// TIA Portal V17 export
// export: Created 2022-11-28T05:31:03.7953951Z, ExportSetting WithDefaults, DisplayName Totally Integrated Automation Portal, DisplayVersion V17, DisplayName TIA Portal Openness, DisplayVersion V17, DisplayName TIA Portal Version Control Interface, DisplayVersion V17, DisplayName STEP 7 Professional, DisplayVersion V17, DisplayName STEP 7 Safety, DisplayVersion V17, DisplayName WinCC Professional, DisplayVersion V17
FUNCTION_BLOCK "MultiProcessing_FB"   // FB2, LAD
{ S7_Optimized_Access := 'TRUE' }
VERSION : 0.1
// stored: AutoNumber true, IsIECCheckEnabled false, IsRetainMemResEnabled false, MemoryReserve 100, SetENOAutomatically false, UDAEnableTagReadback false
   VAR_INPUT
      Start : Bool;
      Reset : Bool;
      RefSwitchTurnTable_PosVac : Bool;
      RefSwitchTurnTable_PosBelt : Bool;
      RefSwitchTurnTable_PosSaw : Bool;
      RefSwitchVac_PosTurnTable : Bool;
      RefSwitchVac_PosOven : Bool;
      RefSwitchOven_FeederInside : Bool;
      RefSwitchOven_FeederOutside : Bool;
      LightBarrierOven : Bool;
      LightBarrierEndOfConBelt : Bool;
   END_VAR
   VAR_OUTPUT
      M2_ConveyorBeltForward : Bool;
      M3_Saw : Bool;
      M4_OvenFeederRetract : Bool;
      M4_OvenFeederExtend : Bool;
      LightOven : Bool;
      PWM_TurnTable : Int;
      PWM_Vacuum : Int;
      Compressor : Bool := true;
   END_VAR
   VAR_IN_OUT
      M1_TurnTableClockwise : Bool;
      M1_TurnTableCounterclockwise : Bool;
      M5_VacuumTowardsOven : Bool;
      M5_VacuumTowardsTurnTable : Bool;
      ValveVacuum : Bool;
      ValveLowering : Bool;
      ValveOvenDoor : Bool;
      ValveFeeder : Bool;
   END_VAR
   VAR
      FeederLoaded : Bool;
      Step_Oven : Int := 0;
      Step_Vacuum : Int := 0;
      Step_TurnTable : Int := 0;
      OpenOvenDoor0 : Bool;
      OpenOvenDoor1 : Bool;
      OpenOvenDoor2 : Bool;
      CloseOvenDoor : Bool;
      Lower0 : Bool;
      Lower1 : Bool;
      Rise0 : Bool;
      Rise1 : Bool;
      Rise2 : Bool;
      M2_TurnTableClockwise : Bool;
      M3_TurnTableClockwise : Bool;
      ActivateVacuum0 : Bool;
      ActivateVacuum1 : Bool;
      DeactivateVacuum : Bool;
      IEC_Timer_LoweringDown { S7_SetPoint := 'True'} : IEC_TIMER;
      IEC_Timer_VacuumOn { S7_SetPoint := 'True'} : IEC_TIMER;
      IEC_Timer_LoweringUp { S7_SetPoint := 'True'} : IEC_TIMER;
      IEC_Timer_VacuumOff { S7_SetPoint := 'True'} : IEC_TIMER;
      IEC_Timer_OvenClose { S7_SetPoint := 'True'} : IEC_TIMER;
      IEC_Timer_OvenLight { S7_SetPoint := 'True'} : IEC_TIMER;
      IEC_Timer_OvenOpen { S7_SetPoint := 'True'} : IEC_TIMER;
      IEC_Timer_Saw { S7_SetPoint := 'True'} : IEC_TIMER;
      IEC_Timer_Onloading { S7_SetPoint := 'True'} : TON_TIME;
      IEC_Timer_Offloading { S7_SetPoint := 'True'} : TON_TIME;
      IEC_Timer_LoweringDownOnOven { S7_SetPoint := 'True'} : TON_TIME;
      IEC_Timer_LoweringUpOffOven { S7_SetPoint := 'True'} : TON_TIME;
      IEC_Timer_OvenReset { S7_SetPoint := 'True'} : TON_TIME;
      IEC_Timer_TurnTablePush { S7_SetPoint := 'True'} : TON_TIME;
      IEC_Timer_DeactivateConveyorBelt { S7_SetPoint := 'True'} : TOF_TIME;
      IEC_Timer_0_Instance { S7_SetPoint := 'True'} : TOF_TIME;
   END_VAR
   VAR_TEMP   // added for the SCL form of the ladder/FBD networks
      _w1 : Bool;
   END_VAR
BEGIN

REGION Network 1: Start/Stop
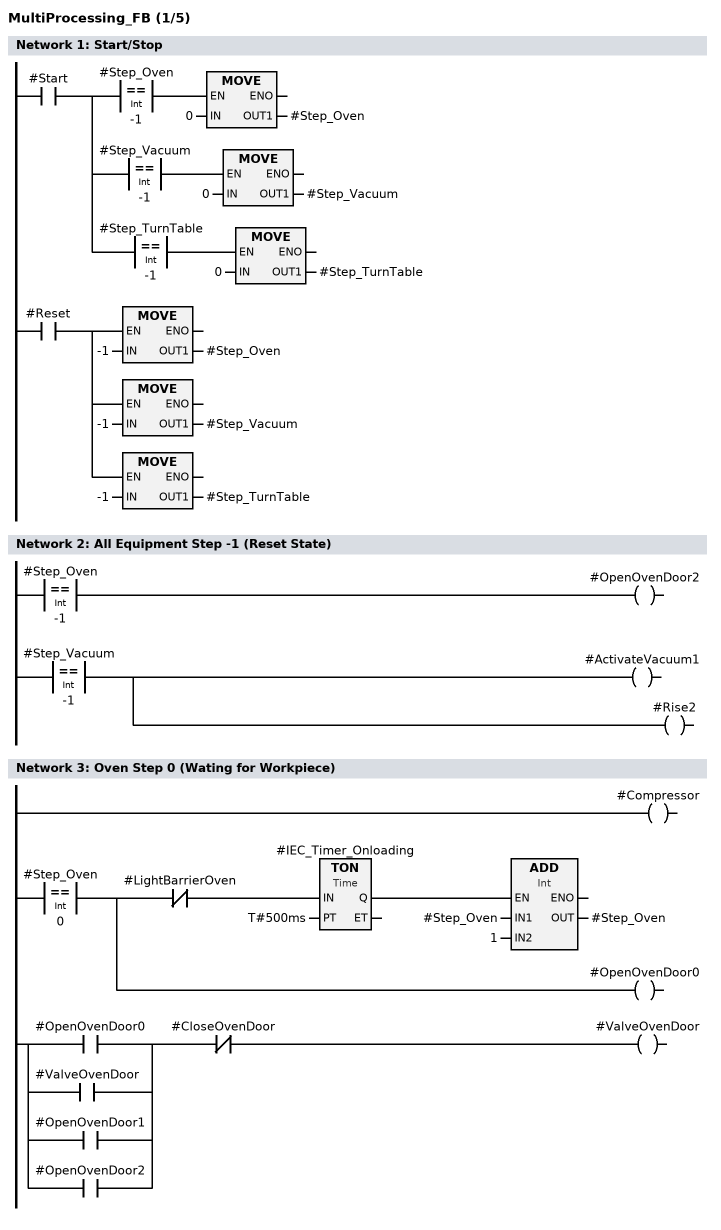
   RUNG wire#powerrail
      Contact( #Start )
      wire#w1
      { S7_Templates := "SrcType := Int" } EQ_Contact(in1 := #Step_Oven, in2 := -1)
      Move(in := 0, out1 => #Step_Oven)
   END_RUNG
   RUNG wire#w1
      { S7_Templates := "SrcType := Int" } EQ_Contact(in1 := #Step_Vacuum, in2 := -1)
      Move(in := 0, out1 => #Step_Vacuum)
   END_RUNG
   RUNG wire#w1
      { S7_Templates := "SrcType := Int" } EQ_Contact(in1 := #Step_TurnTable, in2 := -1)
      Move(in := 0, out1 => #Step_TurnTable)
   END_RUNG
   RUNG wire#powerrail
      Contact( #Reset )
      wire#w2
      Move(in := -1, out1 => #Step_Oven)
   END_RUNG
   RUNG wire#w2
      Move(in := -1, out1 => #Step_Vacuum)
   END_RUNG
   RUNG wire#w2
      Move(in := -1, out1 => #Step_TurnTable)
   END_RUNG
   // the same network as SCL:
   IF #Start AND (#Step_Oven = (-1)) THEN #Step_Oven := 0; END_IF;
   IF #Start AND (#Step_Vacuum = (-1)) THEN #Step_Vacuum := 0; END_IF;
   IF #Start AND (#Step_TurnTable = (-1)) THEN #Step_TurnTable := 0; END_IF;
   IF #Reset THEN
       #Step_Oven := -1;
       #Step_Vacuum := -1;
       #Step_TurnTable := -1;
   END_IF;
END_REGION

REGION Network 2: All Equipment Step -1 (Reset State)
   RUNG wire#powerrail
      { S7_Templates := "SrcType := Int" } EQ_Contact(in1 := #Step_Oven, in2 := -1)
      Coil( #OpenOvenDoor2 )
   END_RUNG
   RUNG wire#powerrail
      { S7_Templates := "SrcType := Int" } EQ_Contact(in1 := #Step_Vacuum, in2 := -1)
      wire#w1
      Coil( #ActivateVacuum1 )
   END_RUNG
   RUNG wire#w1
      Coil( #Rise2 )
   END_RUNG
   // the same network as SCL:
   #OpenOvenDoor2 := #Step_Oven = (-1);
   #ActivateVacuum1 := #Step_Vacuum = (-1);
   #Rise2 := #ActivateVacuum1;
END_REGION

REGION Network 3: Oven Step 0 (Wating for Workpiece)
   RUNG wire#powerrail
      Coil( #Compressor )
   END_RUNG
   RUNG wire#powerrail
      { S7_Templates := "SrcType := Int" } EQ_Contact(in1 := #Step_Oven, in2 := 0)
      wire#w1
      I_Contact( #LightBarrierOven )
      { S7_Templates := "time_type := Time" } #IEC_Timer_Onloading.TON(pt := T#500ms, et =>)
      { S7_Templates := "SrcType := Int" } Add(in1 := #Step_Oven, in2 := 1, out => #Step_Oven)
   END_RUNG
   RUNG wire#w1
      Coil( #OpenOvenDoor0 )
   END_RUNG
   RUNG wire#powerrail
      Contact( #OpenOvenDoor0 )
      wire#w2
      I_Contact( #CloseOvenDoor )
      Coil( #ValveOvenDoor )
   END_RUNG
   RUNG wire#powerrail
      Contact( #ValveOvenDoor )
   END_RUNG wire#w2
   RUNG wire#powerrail
      Contact( #OpenOvenDoor1 )
   END_RUNG wire#w2
   RUNG wire#powerrail
      Contact( #OpenOvenDoor2 )
   END_RUNG wire#w2
   // the same network as SCL:
   #Compressor := TRUE;
   #_w1 := #Step_Oven = 0;
   #IEC_Timer_Onloading(IN := #_w1 AND NOT #LightBarrierOven, PT := T#500ms);   // TON
   IF #IEC_Timer_Onloading.Q THEN #Step_Oven := #Step_Oven + 1; END_IF;
   #OpenOvenDoor0 := #_w1;
   #ValveOvenDoor := (#OpenOvenDoor0 OR #ValveOvenDoor OR #OpenOvenDoor1 OR #OpenOvenDoor2) AND NOT #CloseOvenDoor;
END_REGION

REGION Network 4: Oven Step 1 (Retract and Close Door)
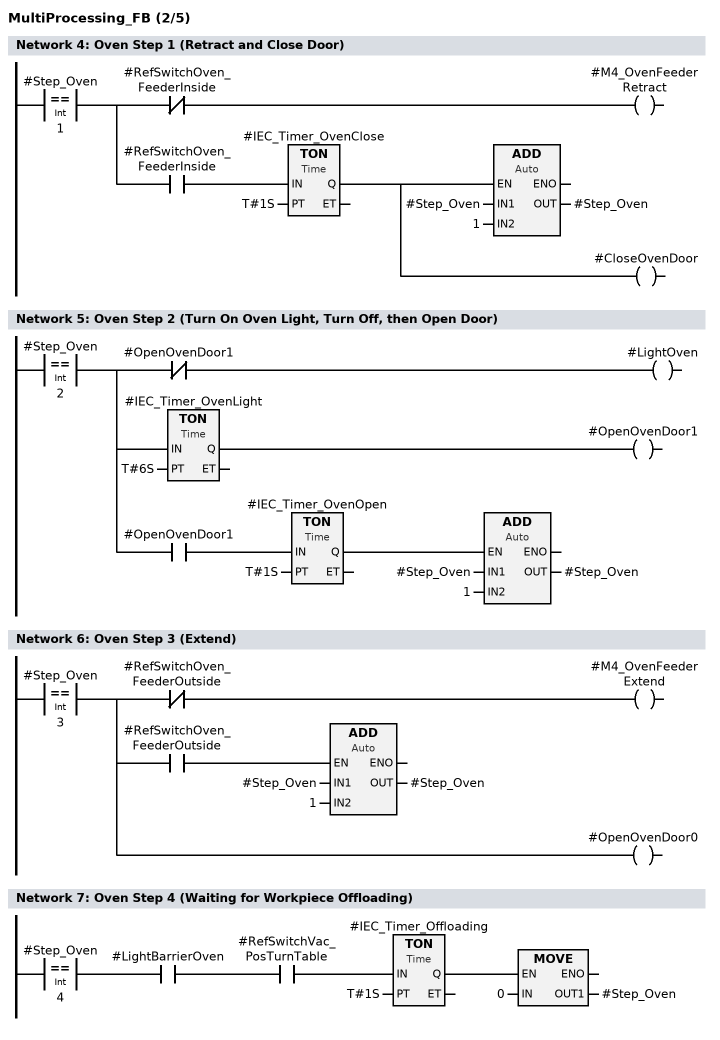
   RUNG wire#powerrail
      { S7_Templates := "SrcType := Int" } EQ_Contact(in1 := #Step_Oven, in2 := 1)
      wire#w1
      I_Contact( #RefSwitchOven_FeederInside )
      Coil( #M4_OvenFeederRetract )
   END_RUNG
   RUNG wire#w1
      Contact( #RefSwitchOven_FeederInside )
      { S7_Templates := "time_type := Time" } #IEC_Timer_OvenClose.TON(pt := T#1S, et =>)
      wire#w2
      Add(in1 := #Step_Oven, in2 := 1, out => #Step_Oven)
   END_RUNG
   RUNG wire#w2
      Coil( #CloseOvenDoor )
   END_RUNG
   // the same network as SCL:
   #_w1 := #Step_Oven = 1;
   #M4_OvenFeederRetract := #_w1 AND NOT #RefSwitchOven_FeederInside;
   #IEC_Timer_OvenClose.TON(IN := #_w1 AND #RefSwitchOven_FeederInside, PT := T#1S);
   IF #IEC_Timer_OvenClose.Q THEN #Step_Oven := #Step_Oven + 1; END_IF;
   #CloseOvenDoor := #IEC_Timer_OvenClose.Q;
END_REGION

REGION Network 5: Oven Step 2 (Turn On Oven Light, Turn Off, then Open Door)
   RUNG wire#powerrail
      { S7_Templates := "SrcType := Int" } EQ_Contact(in1 := #Step_Oven, in2 := 2)
      wire#w1
      I_Contact( #OpenOvenDoor1 )
      Coil( #LightOven )
   END_RUNG
   RUNG wire#w1
      { S7_Templates := "time_type := Time" } #IEC_Timer_OvenLight.TON(pt := T#6S, et =>)
      Coil( #OpenOvenDoor1 )
   END_RUNG
   RUNG wire#w1
      Contact( #OpenOvenDoor1 )
      { S7_Templates := "time_type := Time" } #IEC_Timer_OvenOpen.TON(pt := T#1S, et =>)
      Add(in1 := #Step_Oven, in2 := 1, out => #Step_Oven)
   END_RUNG
   // the same network as SCL:
   #_w1 := #Step_Oven = 2;
   #LightOven := #_w1 AND NOT #OpenOvenDoor1;
   #IEC_Timer_OvenLight.TON(IN := #_w1, PT := T#6S);
   #OpenOvenDoor1 := #IEC_Timer_OvenLight.Q;
   #IEC_Timer_OvenOpen.TON(IN := #_w1 AND #OpenOvenDoor1, PT := T#1S);
   IF #IEC_Timer_OvenOpen.Q THEN #Step_Oven := #Step_Oven + 1; END_IF;
END_REGION

REGION Network 6: Oven Step 3 (Extend)
   RUNG wire#powerrail
      { S7_Templates := "SrcType := Int" } EQ_Contact(in1 := #Step_Oven, in2 := 3)
      wire#w1
      I_Contact( #RefSwitchOven_FeederOutside )
      Coil( #M4_OvenFeederExtend )
   END_RUNG
   RUNG wire#w1
      Contact( #RefSwitchOven_FeederOutside )
      Add(in1 := #Step_Oven, in2 := 1, out => #Step_Oven)
   END_RUNG
   RUNG wire#w1
      Coil( #OpenOvenDoor0 )
   END_RUNG
   // the same network as SCL:
   #_w1 := #Step_Oven = 3;
   #M4_OvenFeederExtend := #_w1 AND NOT #RefSwitchOven_FeederOutside;
   IF #_w1 AND #RefSwitchOven_FeederOutside THEN #Step_Oven := #Step_Oven + 1; END_IF;
   #OpenOvenDoor0 := #_w1;
END_REGION

REGION Network 7: Oven Step 4 (Waiting for Workpiece Offloading)
   RUNG wire#powerrail
      { S7_Templates := "SrcType := Int" } EQ_Contact(in1 := #Step_Oven, in2 := 4)
      Contact( #LightBarrierOven )
      Contact( #RefSwitchVac_PosTurnTable )
      { S7_Templates := "time_type := Time" } #IEC_Timer_Offloading.TON(pt := T#1S, et =>)
      Move(in := 0, out1 => #Step_Oven)
   END_RUNG
   // the same network as SCL:
   #IEC_Timer_Offloading(IN := (#Step_Oven = 4) AND #LightBarrierOven AND #RefSwitchVac_PosTurnTable,   // TON
                         PT := T#1S);
   IF #IEC_Timer_Offloading.Q THEN #Step_Oven := 0; END_IF;
END_REGION

REGION Network 8: Vacuum Step 0 (Move Towards Oven if Possible, Then Wait for Oven Process to Finish)
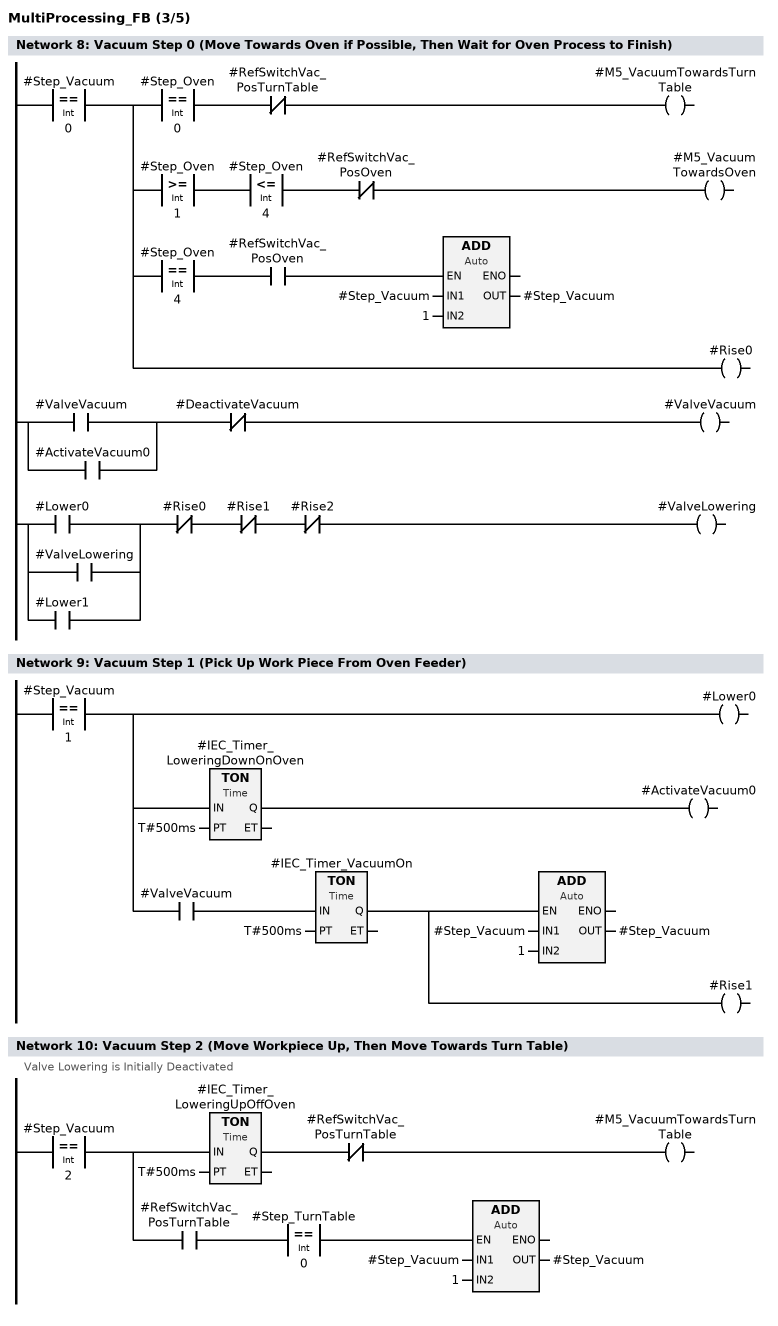
   RUNG wire#powerrail
      { S7_Templates := "SrcType := Int" } EQ_Contact(in1 := #Step_Vacuum, in2 := 0)
      wire#w1
      { S7_Templates := "SrcType := Int" } EQ_Contact(in1 := #Step_Oven, in2 := 0)
      I_Contact( #RefSwitchVac_PosTurnTable )
      Coil( #M5_VacuumTowardsTurnTable )
   END_RUNG
   RUNG wire#w1
      { S7_Templates := "SrcType := Int" } GE_Contact(in1 := #Step_Oven, in2 := 1)
      { S7_Templates := "SrcType := Int" } LE_Contact(in1 := #Step_Oven, in2 := 4)
      I_Contact( #RefSwitchVac_PosOven )
      Coil( #M5_VacuumTowardsOven )
   END_RUNG
   RUNG wire#w1
      { S7_Templates := "SrcType := Int" } EQ_Contact(in1 := #Step_Oven, in2 := 4)
      Contact( #RefSwitchVac_PosOven )
      Add(in1 := #Step_Vacuum, in2 := 1, out => #Step_Vacuum)
   END_RUNG
   RUNG wire#w1
      Coil( #Rise0 )
   END_RUNG
   RUNG wire#powerrail
      Contact( #ValveVacuum )
      wire#w2
      I_Contact( #DeactivateVacuum )
      Coil( #ValveVacuum )
   END_RUNG
   RUNG wire#powerrail
      Contact( #ActivateVacuum0 )
   END_RUNG wire#w2
   RUNG wire#powerrail
      Contact( #Lower0 )
      wire#w3
      I_Contact( #Rise0 )
      I_Contact( #Rise1 )
      I_Contact( #Rise2 )
      Coil( #ValveLowering )
   END_RUNG
   RUNG wire#powerrail
      Contact( #ValveLowering )
   END_RUNG wire#w3
   RUNG wire#powerrail
      Contact( #Lower1 )
   END_RUNG wire#w3
   // the same network as SCL:
   #_w1 := #Step_Vacuum = 0;
   #M5_VacuumTowardsTurnTable := #_w1 AND (#Step_Oven = 0) AND NOT #RefSwitchVac_PosTurnTable;
   #M5_VacuumTowardsOven := #_w1 AND (#Step_Oven >= 1) AND (#Step_Oven <= 4) AND NOT #RefSwitchVac_PosOven;
   IF #_w1 AND (#Step_Oven = 4) AND #RefSwitchVac_PosOven THEN #Step_Vacuum := #Step_Vacuum + 1; END_IF;
   #Rise0 := #_w1;
   #ValveVacuum := (#ValveVacuum OR #ActivateVacuum0) AND NOT #DeactivateVacuum;
   #ValveLowering := (#Lower0 OR #ValveLowering OR #Lower1) AND NOT #Rise0 AND NOT #Rise1 AND NOT #Rise2;
END_REGION

REGION Network 9: Vacuum Step 1 (Pick Up Work Piece From Oven Feeder)
   RUNG wire#powerrail
      { S7_Templates := "SrcType := Int" } EQ_Contact(in1 := #Step_Vacuum, in2 := 1)
      wire#w1
      Coil( #Lower0 )
   END_RUNG
   RUNG wire#w1
      { S7_Templates := "time_type := Time" } #IEC_Timer_LoweringDownOnOven.TON(pt := T#500ms, et =>)
      Coil( #ActivateVacuum0 )
   END_RUNG
   RUNG wire#w1
      Contact( #ValveVacuum )
      { S7_Templates := "time_type := Time" } #IEC_Timer_VacuumOn.TON(pt := T#500ms, et =>)
      wire#w2
      Add(in1 := #Step_Vacuum, in2 := 1, out => #Step_Vacuum)
   END_RUNG
   RUNG wire#w2
      Coil( #Rise1 )
   END_RUNG
   // the same network as SCL:
   #Lower0 := #Step_Vacuum = 1;
   #IEC_Timer_LoweringDownOnOven(IN := #Lower0, PT := T#500ms);   // TON
   #ActivateVacuum0 := #IEC_Timer_LoweringDownOnOven.Q;
   #IEC_Timer_VacuumOn.TON(IN := #Lower0 AND #ValveVacuum, PT := T#500ms);
   IF #IEC_Timer_VacuumOn.Q THEN #Step_Vacuum := #Step_Vacuum + 1; END_IF;
   #Rise1 := #IEC_Timer_VacuumOn.Q;
END_REGION

REGION Network 10: Vacuum Step 2 (Move Workpiece Up, Then Move Towards Turn Table)
   // Valve Lowering is Initially Deactivated
   RUNG wire#powerrail
      { S7_Templates := "SrcType := Int" } EQ_Contact(in1 := #Step_Vacuum, in2 := 2)
      wire#w1
      { S7_Templates := "time_type := Time" } #IEC_Timer_LoweringUpOffOven.TON(pt := T#500ms, et =>)
      I_Contact( #RefSwitchVac_PosTurnTable )
      Coil( #M5_VacuumTowardsTurnTable )
   END_RUNG
   RUNG wire#w1
      Contact( #RefSwitchVac_PosTurnTable )
      { S7_Templates := "SrcType := Int" } EQ_Contact(in1 := #Step_TurnTable, in2 := 0)
      Add(in1 := #Step_Vacuum, in2 := 1, out => #Step_Vacuum)
   END_RUNG
   // the same network as SCL:
   #_w1 := #Step_Vacuum = 2;
   #IEC_Timer_LoweringUpOffOven(IN := #_w1, PT := T#500ms);   // TON
   #M5_VacuumTowardsTurnTable := #IEC_Timer_LoweringUpOffOven.Q AND NOT #RefSwitchVac_PosTurnTable;
   IF #_w1 AND #RefSwitchVac_PosTurnTable AND (#Step_TurnTable = 0) THEN
       #Step_Vacuum := #Step_Vacuum + 1;
   END_IF;
END_REGION

REGION Network 11: Vacuum Step 3 (Lower Workpiece unto Turn Table)
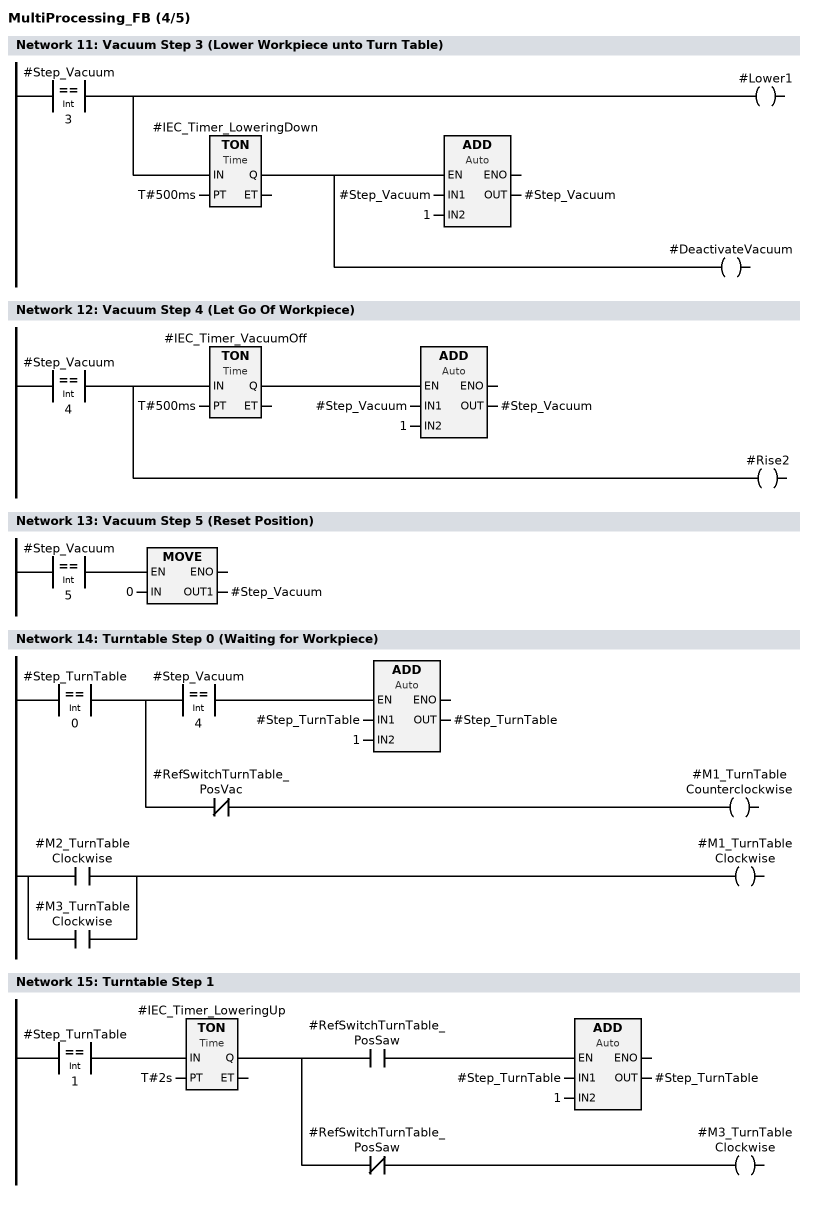
   RUNG wire#powerrail
      { S7_Templates := "SrcType := Int" } EQ_Contact(in1 := #Step_Vacuum, in2 := 3)
      wire#w1
      Coil( #Lower1 )
   END_RUNG
   RUNG wire#w1
      { S7_Templates := "time_type := Time" } #IEC_Timer_LoweringDown.TON(pt := T#500ms, et =>)
      wire#w2
      Add(in1 := #Step_Vacuum, in2 := 1, out => #Step_Vacuum)
   END_RUNG
   RUNG wire#w2
      Coil( #DeactivateVacuum )
   END_RUNG
   // the same network as SCL:
   #Lower1 := #Step_Vacuum = 3;
   #IEC_Timer_LoweringDown.TON(IN := #Lower1, PT := T#500ms);
   IF #IEC_Timer_LoweringDown.Q THEN #Step_Vacuum := #Step_Vacuum + 1; END_IF;
   #DeactivateVacuum := #IEC_Timer_LoweringDown.Q;
END_REGION

REGION Network 12: Vacuum Step 4 (Let Go Of Workpiece)
   RUNG wire#powerrail
      { S7_Templates := "SrcType := Int" } EQ_Contact(in1 := #Step_Vacuum, in2 := 4)
      wire#w1
      { S7_Templates := "time_type := Time" } #IEC_Timer_VacuumOff.TON(pt := T#500ms, et =>)
      Add(in1 := #Step_Vacuum, in2 := 1, out => #Step_Vacuum)
   END_RUNG
   RUNG wire#w1
      Coil( #Rise2 )
   END_RUNG
   // the same network as SCL:
   #_w1 := #Step_Vacuum = 4;
   #IEC_Timer_VacuumOff.TON(IN := #_w1, PT := T#500ms);
   IF #IEC_Timer_VacuumOff.Q THEN #Step_Vacuum := #Step_Vacuum + 1; END_IF;
   #Rise2 := #_w1;
END_REGION

REGION Network 13: Vacuum Step 5 (Reset Position)
   RUNG wire#powerrail
      { S7_Templates := "SrcType := Int" } EQ_Contact(in1 := #Step_Vacuum, in2 := 5)
      Move(in := 0, out1 => #Step_Vacuum)
   END_RUNG
   // the same network as SCL:
   IF #Step_Vacuum = 5 THEN #Step_Vacuum := 0; END_IF;
END_REGION

REGION Network 14: Turntable Step 0 (Waiting for Workpiece)
   RUNG wire#powerrail
      { S7_Templates := "SrcType := Int" } EQ_Contact(in1 := #Step_TurnTable, in2 := 0)
      wire#w1
      { S7_Templates := "SrcType := Int" } EQ_Contact(in1 := #Step_Vacuum, in2 := 4)
      Add(in1 := #Step_TurnTable, in2 := 1, out => #Step_TurnTable)
   END_RUNG
   RUNG wire#w1
      I_Contact( #RefSwitchTurnTable_PosVac )
      Coil( #M1_TurnTableCounterclockwise )
   END_RUNG
   RUNG wire#powerrail
      Contact( #M2_TurnTableClockwise )
      wire#w2
      Coil( #M1_TurnTableClockwise )
   END_RUNG
   RUNG wire#powerrail
      Contact( #M3_TurnTableClockwise )
   END_RUNG wire#w2
   // the same network as SCL:
   #_w1 := #Step_TurnTable = 0;
   IF #_w1 AND (#Step_Vacuum = 4) THEN #Step_TurnTable := #Step_TurnTable + 1; END_IF;
   #M1_TurnTableCounterclockwise := #_w1 AND NOT #RefSwitchTurnTable_PosVac;
   #M1_TurnTableClockwise := #M2_TurnTableClockwise OR #M3_TurnTableClockwise;
END_REGION

REGION Network 15: Turntable Step 1
   RUNG wire#powerrail
      { S7_Templates := "SrcType := Int" } EQ_Contact(in1 := #Step_TurnTable, in2 := 1)
      { S7_Templates := "time_type := Time" } #IEC_Timer_LoweringUp.TON(pt := T#2s, et =>)
      wire#w1
      Contact( #RefSwitchTurnTable_PosSaw )
      Add(in1 := #Step_TurnTable, in2 := 1, out => #Step_TurnTable)
   END_RUNG
   RUNG wire#w1
      I_Contact( #RefSwitchTurnTable_PosSaw )
      Coil( #M3_TurnTableClockwise )
   END_RUNG
   // the same network as SCL:
   #IEC_Timer_LoweringUp.TON(IN := #Step_TurnTable = 1, PT := T#2s);
   IF #IEC_Timer_LoweringUp.Q AND #RefSwitchTurnTable_PosSaw THEN
       #Step_TurnTable := #Step_TurnTable + 1;
   END_IF;
   #M3_TurnTableClockwise := #IEC_Timer_LoweringUp.Q AND NOT #RefSwitchTurnTable_PosSaw;
END_REGION

REGION Network 16: Turntable Step 2
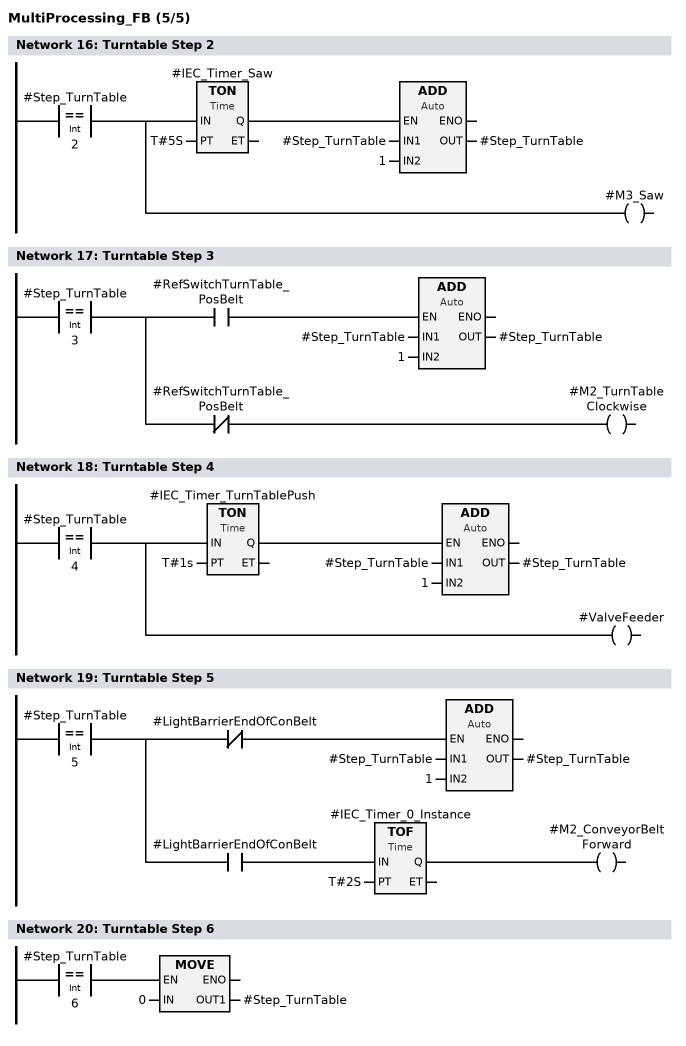
   RUNG wire#powerrail
      { S7_Templates := "SrcType := Int" } EQ_Contact(in1 := #Step_TurnTable, in2 := 2)
      wire#w1
      { S7_Templates := "time_type := Time" } #IEC_Timer_Saw.TON(pt := T#5S, et =>)
      Add(in1 := #Step_TurnTable, in2 := 1, out => #Step_TurnTable)
   END_RUNG
   RUNG wire#w1
      Coil( #M3_Saw )
   END_RUNG
   // the same network as SCL:
   #_w1 := #Step_TurnTable = 2;
   #IEC_Timer_Saw.TON(IN := #_w1, PT := T#5S);
   IF #IEC_Timer_Saw.Q THEN #Step_TurnTable := #Step_TurnTable + 1; END_IF;
   #M3_Saw := #_w1;
END_REGION

REGION Network 17: Turntable Step 3
   RUNG wire#powerrail
      { S7_Templates := "SrcType := Int" } EQ_Contact(in1 := #Step_TurnTable, in2 := 3)
      wire#w1
      Contact( #RefSwitchTurnTable_PosBelt )
      Add(in1 := #Step_TurnTable, in2 := 1, out => #Step_TurnTable)
   END_RUNG
   RUNG wire#w1
      I_Contact( #RefSwitchTurnTable_PosBelt )
      Coil( #M2_TurnTableClockwise )
   END_RUNG
   // the same network as SCL:
   #_w1 := #Step_TurnTable = 3;
   IF #_w1 AND #RefSwitchTurnTable_PosBelt THEN #Step_TurnTable := #Step_TurnTable + 1; END_IF;
   #M2_TurnTableClockwise := #_w1 AND NOT #RefSwitchTurnTable_PosBelt;
END_REGION

REGION Network 18: Turntable Step 4
   RUNG wire#powerrail
      { S7_Templates := "SrcType := Int" } EQ_Contact(in1 := #Step_TurnTable, in2 := 4)
      wire#w1
      { S7_Templates := "time_type := Time" } #IEC_Timer_TurnTablePush.TON(pt := T#1s, et =>)
      Add(in1 := #Step_TurnTable, in2 := 1, out => #Step_TurnTable)
   END_RUNG
   RUNG wire#w1
      Coil( #ValveFeeder )
   END_RUNG
   // the same network as SCL:
   #_w1 := #Step_TurnTable = 4;
   #IEC_Timer_TurnTablePush(IN := #_w1, PT := T#1s);   // TON
   IF #IEC_Timer_TurnTablePush.Q THEN #Step_TurnTable := #Step_TurnTable + 1; END_IF;
   #ValveFeeder := #_w1;
END_REGION

REGION Network 19: Turntable Step 5
   RUNG wire#powerrail
      { S7_Templates := "SrcType := Int" } EQ_Contact(in1 := #Step_TurnTable, in2 := 5)
      wire#w1
      I_Contact( #LightBarrierEndOfConBelt )
      Add(in1 := #Step_TurnTable, in2 := 1, out => #Step_TurnTable)
   END_RUNG
   RUNG wire#w1
      Contact( #LightBarrierEndOfConBelt )
      { S7_Templates := "time_type := Time" } #IEC_Timer_0_Instance.TOF(pt := T#2S, et =>)
      Coil( #M2_ConveyorBeltForward )
   END_RUNG
   // the same network as SCL:
   #_w1 := #Step_TurnTable = 5;
   IF #_w1 AND NOT #LightBarrierEndOfConBelt THEN #Step_TurnTable := #Step_TurnTable + 1; END_IF;
   #IEC_Timer_0_Instance(IN := #_w1 AND #LightBarrierEndOfConBelt, PT := T#2S);   // TOF
   #M2_ConveyorBeltForward := #IEC_Timer_0_Instance.Q;
END_REGION

REGION Network 20: Turntable Step 6
   RUNG wire#powerrail
      { S7_Templates := "SrcType := Int" } EQ_Contact(in1 := #Step_TurnTable, in2 := 6)
      Move(in := 0, out1 => #Step_TurnTable)
   END_RUNG
   // the same network as SCL:
   IF #Step_TurnTable = 6 THEN #Step_TurnTable := 0; END_IF;
END_REGION
END_FUNCTION_BLOCK
